// TIA Portal project "HMI_denGiaoThong_T3" (V14)

(* hardware
DEVICE "S7-1200 station_1"  S7-1200 Station
   slot 0: "Rack_0"  S7-1200 Rack  Rack  V1.0
   slot 1: "PLC_1"  CPU 1214C DC/DC/DC  6ES7 214-1AG40-0XB0  V4.2
DEVICE "HMI_1"  KTP700 Basic PN
   slot 0: "KTP700 Basic PN"  KTP700 Basic PN  6AV2 123-2GB03-0AX0  14.0.1.0
   slot 1: "HMI_RT_1"  KTP700 Basic PN  6AV2 123-2GB03-0AX0  14.0.1.0
   slot 5: "HMI_1.IE_CP_1"  PROFINET Interface  14.0.1.0
      slot 1: "PROFINET Interface_1"  PROFINET Interface
         slot 1: "Port_1"  Port
*)

// ===== PLC "PLC_1"  CPU 1214C DC/DC/DC =====

VAR_GLOBAL   // PLC tag table "Default tag table"
   "UT1" AT %M0.0 : Bool;
   "D1" AT %Q0.0 : Bool;
   "X1" AT %Q0.1 : Bool;
   "D2" AT %Q0.2 : Bool;
   "UT2" AT %M0.1 : Bool;
   "X2" AT %Q0.3 : Bool;
   "CT_V" AT %M0.2 : Bool;
   "V1" AT %Q0.4 : Bool;
   "V2" AT %Q0.5 : Bool;
END_VAR

// folder: System blocks/Program resources

DATA_BLOCK "hkh"   // DB1
{ S7_Optimized_Access := 'TRUE' }
AUTHOR : Simatic
FAMILY : IEC
NAME : IEC_TMR
VERSION : 1.0
// stored: InstanceOfName IEC_TIMER
"IEC_TIMER"
BEGIN
END_DATA_BLOCK

DATA_BLOCK "IEC_Tmer_0_DB_1"   // DB2
{ S7_Optimized_Access := 'TRUE' }
AUTHOR : Simatic
FAMILY : IEC
NAME : IEC_TMR
VERSION : 1.0
// stored: InstanceOfName IEC_TIMER
"IEC_TIMER"
BEGIN
END_DATA_BLOCK

DATA_BLOCK "IEC_Time_0_DB_2"   // DB3
{ S7_Optimized_Access := 'TRUE' }
AUTHOR : Simatic
FAMILY : IEC
NAME : IEC_TMR
VERSION : 1.0
// stored: InstanceOfName IEC_TIMER
"IEC_TIMER"
BEGIN
END_DATA_BLOCK

DATA_BLOCK "IEC_Timer0_DB_3"   // DB4
{ S7_Optimized_Access := 'TRUE' }
AUTHOR : Simatic
FAMILY : IEC
NAME : IEC_TMR
VERSION : 1.0
// stored: InstanceOfName IEC_TIMER
"IEC_TIMER"
BEGIN
END_DATA_BLOCK

DATA_BLOCK "IECTimer_0_DB_4"   // DB5
{ S7_Optimized_Access := 'TRUE' }
AUTHOR : Simatic
FAMILY : IEC
NAME : IEC_TMR
VERSION : 1.0
// stored: InstanceOfName IEC_TIMER
"IEC_TIMER"
BEGIN
END_DATA_BLOCK

DATA_BLOCK "IECTimer_0_DB_5"   // DB6
{ S7_Optimized_Access := 'TRUE' }
AUTHOR : Simatic
FAMILY : IEC
NAME : IEC_TMR
VERSION : 1.0
// stored: InstanceOfName IEC_TIMER
"IEC_TIMER"
BEGIN
END_DATA_BLOCK

// folder: (top level)

ORGANIZATION_BLOCK "Main"   // OB1, LAD, ProgramCycle
TITLE = "Main Program Sweep (Cycle)"
{ S7_Optimized_Access := 'TRUE' }
VERSION : 0.1
   VAR_INPUT
      Initial_Call : Bool;   // Initial call of this OB
      Remanence : Bool;   // =True, if remanent data are available
   END_VAR
   VAR_TEMP   // added for the SCL form of the ladder/FBD networks
      _w1 : Bool;
   END_VAR
BEGIN

REGION Network 1
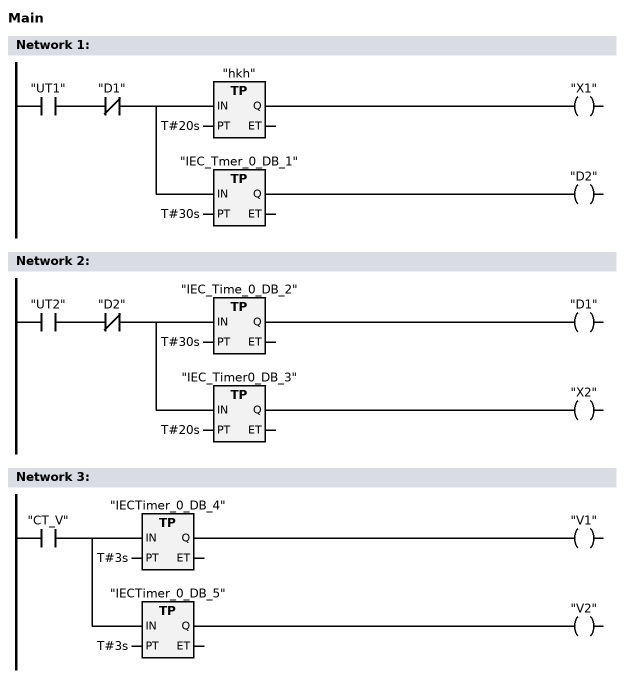
   #_w1 := "UT1" AND NOT "D1";
   "hkh".TP(IN := #_w1, PT := T#20s);
   "X1" := "hkh".Q;
   "IEC_Tmer_0_DB_1".TP(IN := #_w1, PT := T#30s);
   "D2" := "IEC_Tmer_0_DB_1".Q;
END_REGION

REGION Network 2
   #_w1 := "UT2" AND NOT "D2";
   "IEC_Time_0_DB_2".TP(IN := #_w1, PT := T#30s);
   "D1" := "IEC_Time_0_DB_2".Q;
   "IEC_Timer0_DB_3".TP(IN := #_w1, PT := T#20s);
   "X2" := "IEC_Timer0_DB_3".Q;
END_REGION

REGION Network 3
   "IECTimer_0_DB_4".TP(IN := "CT_V", PT := T#3s);
   "V1" := "IECTimer_0_DB_4".Q;
   "IECTimer_0_DB_5".TP(IN := "CT_V", PT := T#3s);
   "V2" := "IECTimer_0_DB_5".Q;
END_REGION
END_ORGANIZATION_BLOCK

(* ===== HMI "HMI_RT_1" =====
system functions are stored by id; their names below are inferred from use
connection "HMI_Connection_1": ETHERNET, SMART_S7_1200_OMS

HMI tags "Default tag table"
   "Tag_ScreenNumber" : UInt, internal
   "D2" : Bool = PLC D2 AT %Q0.2, 1 s
   "X2" : Bool = PLC X2 AT %Q0.3, 1 s
   "V2" : Bool = PLC V2 AT %Q0.5, 1 s
   "D1" : Bool = PLC D1 AT %Q0.0, 1 s
   "X1" : Bool = PLC X1 AT %Q0.1, 1 s
   "V1" : Bool = PLC V1 AT %Q0.4, 1 s
   "UT1" : Bool = PLC UT1 AT %M0.0, 1 s
   "UT2" : Bool = PLC UT2 AT %M0.1, 1 s
   "CT_V" : Bool = PLC CT_V AT %M0.2, 1 s

Template "Template_1" 800x480
   Button "Exit" at 714,429 size 71x50; TextOff 'Exit'; PictureOff "ExitRuntime_KTP700_Basic_PN_TR"; PictureOn "ExitRuntime_KTP700_Basic_PN_TR"
      on Release: StopRuntime(0)
   Button "Template_Button" at 614,429 size 71x50; TextOff 'Text'
   Button "Template_Button_1" at 514,429 size 71x50; TextOff 'Text'
   Button "Template_Button_2" at 414,429 size 71x50; TextOff 'Text'
   Button "Template_Button_3" at 314,429 size 71x50; TextOff 'Text'
   Button "Template_Button_4" at 214,429 size 71x50; TextOff 'Text'
   Button "Alarms" at 114,429 size 71x50; TextOff 'Alarms'; PictureOff "AlarmDisplay_KTP700_Basic_PN_TR"; PictureOn "AlarmDisplay_KTP700_Basic_PN_TR"
      on Release: function_ef3f5d25("Alarm window_Unacknowledged", -1)
   Button "Start screen" at 14,429 size 71x50; TextOff 'Start screen'; PictureOff "NavigateHome_KTP700_Basic_PN_TR"; PictureOn "NavigateHome_KTP700_Basic_PN_TR"
      on Release: ActivateScreen("Root screen", 0)
   SymbolicIOField "Symbolic_IO_Field_Screen" at 93,9 size 600x33; TextOff '0'; TextOn '1'; TextList "TextList_ScreenNames"
      ProcessValue <- "Tag_ScreenNumber"
      on Change: ActivateScreenByNumber("Tag_ScreenNumber", 0)
   DateTimeField "HmiScreenItemData" at 695,25 size 105x25
   DateTimeField "HmiScreenItemData_1" at 695,0 size 105x25
   GraphicView "Logo" at 0,0 size 91x51; Picture "Logo of HMI_1"

screen "Root screen" 800x480, template "Template_1"
   on GenerateScreen: SetTag("Tag_ScreenNumber", 1)
   Circle "Circle_4" at 491,77 size 22x22
      Appearance <- "D1"
   Circle "Circle_5" at 491,108 size 22x22
      Appearance <- "X1"
   Circle "Circle_6" at 491,139 size 22x22
      Appearance <- "V1"
   Circle "Circle_10" at 269,319 size 22x22
      Appearance <- "D2"
   Circle "Circle_11" at 269,350 size 22x22
      Appearance <- "X2"
   Circle "Circle_12" at 269,381 size 22x22
      Appearance <- "V2"
   Button "Button_1" at 544,139 size 94x27; TextOff 'UT1'
      on Click: InvertBit("UT1")
      Appearance <- "UT1"
   Button "Button_2" at 145,381 size 94x27; TextOff 'UT2'
      Appearance <- "UT2"
      on Click: InvertBit("UT2")
   Button "Button_3" at 659,356 size 96x32; TextOff 'START'
      Appearance <- "CT_V"
      on Click: InvertBit("CT_V")
*)